INTERFACE I_BaseAxis

PROPERTY ActualPosition : LREAL
GET
END_GET
SET
END_SET
END_PROPERTY

PROPERTY Busy : BOOL
GET
END_GET
END_PROPERTY

PROPERTY Calibrated : BOOL
GET
END_GET
END_PROPERTY

PROPERTY Enable : BOOL
GET
END_GET
SET
END_SET
END_PROPERTY

PROPERTY Error : BOOL
GET
END_GET
END_PROPERTY

PROPERTY ErrorID : UDINT
GET
END_GET
END_PROPERTY

PROPERTY HomeAxis : BOOL
GET
END_GET
SET
END_SET
END_PROPERTY

PROPERTY InNegLimit : BOOL
GET
END_GET
END_PROPERTY

PROPERTY InPosLimit : BOOL
GET
END_GET
END_PROPERTY

PROPERTY MoveNeg : BOOL
GET
END_GET
SET
END_SET
END_PROPERTY

PROPERTY MovePos : BOOL
GET
END_GET
SET
END_SET
END_PROPERTY

PROPERTY Position : LREAL
GET
END_GET
SET
END_SET
END_PROPERTY

PROPERTY Ready : BOOL
GET
END_GET
END_PROPERTY

METHOD Reset : BOOL
VAR_INPUT
END_VAR
END_METHOD

PROPERTY Velocity : LREAL
GET
END_GET
SET
END_SET
END_PROPERTY

END_INTERFACE

(* stored: Version 1.1.0.1, ProductVersion 3.1.4024.15
   Itf I_BaseAxis: Id {b01d5c4d-03ee-40b2-9a40-3d7abce441f2}
   Property ActualPosition: Id {0eda8458-a0f4-4030-bbb2-8516eb7dc1fd}
   Get Get: Id {27227f52-1004-4bfd-85ce-1b8cf5d1caab}
   Set Set: Id {70191a9a-9a0d-48b6-845e-aba3d25e1f3e}
   Property Busy: Id {ba5504aa-3dda-42ca-bac2-51c45207c93a}
   Get Get: Id {b9cb56cd-c171-469f-b53d-6f00d1c9714f}
   Property Calibrated: Id {19e9d110-74bf-4045-a3bf-5f358d99765b}
   Get Get: Id {e5bd9191-9ec2-48a2-8d46-291347e47d6c}
   Property Enable: Id {f00a00ca-cd53-4195-883b-b5305c4bc6dc}
   Get Get: Id {54ded346-e658-4c29-b3c2-795c8c4546ec}
   Set Set: Id {27371135-a06f-4870-87b9-fc5625a5988c}
   Property Error: Id {38bbb32e-3c0a-4087-ba48-cbebfbc23d31}
   Get Get: Id {fb98412b-4dc9-45ea-adcd-7d8dc14c2ef1}
   Property ErrorID: Id {55a37fa5-5d66-4267-aad3-3a98aa372c29}
   Get Get: Id {25802475-7347-42d5-a54f-4b632a030274}
   Property HomeAxis: Id {d1537209-25a2-4e1c-94aa-5e8bec67a977}
   Get Get: Id {9c29ba6a-1a3a-4434-bcdf-2c14e7dc6431}
   Set Set: Id {d3c08ea7-d2cd-4af0-868f-5fadac210a9e}
   Property InNegLimit: Id {7ed5f7ce-2d19-4c51-9235-cf95950da38a}
   Get Get: Id {b2c791f1-a929-476d-b8be-d54029b01049}
   Property InPosLimit: Id {c0bbcafb-ad06-49ef-b33e-162cf573768b}
   Get Get: Id {987fb4b2-a0ed-4b53-9433-3bafe5e57d71}
   Property MoveNeg: Id {273cb633-0163-4c0e-aa79-479108adb62f}
   Get Get: Id {66565ae8-18e2-44be-8013-686e2e637e40}
   Set Set: Id {cb8eec97-cc0f-45c9-80ee-b220687ec4c4}
   Property MovePos: Id {a0bc8eac-5450-447e-b5e2-4ae970562be2}
   Get Get: Id {591ab01b-6e09-472d-ba71-ce72830b3221}
   Set Set: Id {a69c274c-e5d2-4d7f-8117-90ecc821dbc1}
   Property Position: Id {b990da48-4810-4c07-9b89-53062240be15}
   Get Get: Id {4e1c508f-c40a-4af5-9f87-d147eca48a3e}
   Set Set: Id {e09eff94-3fd9-4578-a736-1299b29646c3}
   Property Ready: Id {7d6e258f-d171-42f5-a90b-a905b21fe52c}
   Get Get: Id {910a411c-438b-480a-bf39-34253c3cab2f}
   Method Reset: Id {466c4f7e-e945-477b-a4db-3103979d61bc}
   Property Velocity: Id {ccd581c9-c5ee-4b41-8cf1-7d61f7e80a83}
   Get Get: Id {16838da0-ce65-47be-9f18-f1ac4e6a8893}
   Set Set: Id {685648c2-6602-486f-95c0-65e9bf425878} *)
